// TIA Portal V16 export
// export: Created 2021-03-05T14:22:11.7705928Z, ExportSetting WithDefaults, DisplayName Totally Integrated Automation Portal, DisplayVersion V16, DisplayName TIA Portal Version Control Interface, DisplayVersion V16, DisplayName TIA Portal Openness, DisplayVersion V16, DisplayName SINAMICS Startdrive Advanced, DisplayVersion V16, DisplayName SINAMICS Startdrive G130, G150, S120, S150, SINAMICS MV, S210, DisplayVersion V16, DisplayName SINAMICS Startdrive G110M, G120, G120C, G120D, G120P, DisplayVersion V16, DisplayName STEP 7 Professional, DisplayVersion V16, DisplayName STEP 7 Safety, DisplayVersion V16, DisplayName WinCC Professional, DisplayVersion V16
FUNCTION_BLOCK "fbRack"   // FB3, LAD
{ S7_Optimized_Access := 'TRUE' }
VERSION : 0.1
// stored: AutoNumber true, IsIECCheckEnabled false, IsRetainMemResEnabled false, MemoryReserve 100, SetENOAutomatically false, UDAEnableTagReadback false
   VAR_INPUT
      arrAI { ExternalAccessible := 'False'; ExternalVisible := 'False'; ExternalWritable := 'False'} : Array[1.."NUM_AI_RACK"] of Int;
      AI AT arrAI : "udtRackAI";
   END_VAR
   VAR
      Fertigation : "fbRackFertigation";
   END_VAR
   VAR_TEMP
      i : Int;
   END_VAR
BEGIN

REGION Network 1 (SCL)
   #Fertigation(arrAI := #Fertigation.arrAI,
                arrDQ => #Fertigation.arrDQ);

   // Set rack-level outputs
END_REGION
END_FUNCTION_BLOCK
